///EL2964 | 1-channel digital output terminal, TwinSAFE, 24 V DC, potential-free contacts
FUNCTION_BLOCK EL2964_v0_00

END_FUNCTION_BLOCK

(* stored: Version 1.1.0.1, ProductVersion 3.1.0.25
   POU EL2964_v0_00: Id {da88f501-ef06-4c75-bce9-a89e8f9abd13} *)
